# B&R Automation Studio project MotionTestBenchMaster (part 37)

#### Init.st - Init code
```iecst
PROGRAM _INIT
	(**********************************)
	(*  Mp Link Hierarchy management  *)
	(**********************************)
	fbMpComLinkToParent_Spare		(ParentLink := mpCOM_MAIN, MpLink := ADR(VAR_SpareLink));

	(**********************************)
	(* The machine is the higher Link *)
	(**********************************)
	fbMpComLinkToParent_Machine		(ParentLink := mpCOM_MAIN, MpLink := ADR(VAR_MachineLink));
	fbMpComLinkToParent_Master		(ParentLink := fbMpComLinkToParent_Machine.LinkOut,	MpLink := ADR(VAR_MasterModuleLink));
	fbMpComLinkToParent_Filler		(ParentLink := fbMpComLinkToParent_Machine.LinkOut,	MpLink := ADR(VAR_FillerModuleLink));

	IF VAR_AxOutletMain.nc_obj_inf.node_nr > 0 THEN	//At least the main axis in the outlet module
		fbMpComLinkToParent_Outlet	(ParentLink := fbMpComLinkToParent_Machine.LinkOut,	MpLink := ADR(VAR_OutletModuleLink));
	ELSE
		fbMpComLinkToParent_Outlet	(ParentLink := fbMpComLinkToParent_Spare.LinkOut,	MpLink := ADR(VAR_OutletModuleLink));
	END_IF

	IF VAR_AxInletMain.nc_obj_inf.node_nr > 0 THEN	//At least the main axis in the inlet module
		fbMpComLinkToParent_Inlet	(ParentLink := fbMpComLinkToParent_Machine.LinkOut,	MpLink := ADR(VAR_InletModuleLink));
	ELSE
		fbMpComLinkToParent_Inlet	(ParentLink := fbMpComLinkToParent_Spare.LinkOut,	MpLink := ADR(VAR_InletModuleLink));
	END_IF

	fbMpComLinkToParentAlarmMain	(ParentLink := fbMpComLinkToParent_Machine.LinkOut,	MpLink := ADR(gMainAlarmXCoreLink));

	(**********************************)
	(* Init of Link on Master Module  *)
	(**********************************)
	fbMpComLinkToParent_AlarmXMaster(ParentLink := fbMpComLinkToParent_Master.LinkOut,	MpLink := ADR(gMasterAlarmXCoreLink));
	fbMpComLinkToParent_MasterAxis 	(ParentLink := fbMpComLinkToParent_Master.LinkOut,	MpLink := ADR(gMasterLink));

	IF VAR_AxPowerSupply01.nc_obj_inf.node_nr > 0 THEN
		fbMpComLinkToParent_Pwr01 		(ParentLink := fbMpComLinkToParent_Master.LinkOut,	MpLink := ADR(gMasterPwr01Link));
	ELSE
		fbMpComLinkToParent_Pwr01		(ParentLink := fbMpComLinkToParent_Spare.LinkOut,	MpLink := ADR(gMasterPwr01Link));
	END_IF

	IF VAR_AxPowerSupply02.nc_obj_inf.node_nr > 0 THEN
		fbMpComLinkToParent_Pwr02 		(ParentLink := fbMpComLinkToParent_Master.LinkOut,	MpLink := ADR(gMasterPwr02Link));
	ELSE
		fbMpComLinkToParent_Pwr02 		(ParentLink := fbMpComLinkToParent_Spare.LinkOut,	MpLink := ADR(gMasterPwr02Link));
	END_IF

	(**********************************)
	(* Init of Link on Filler Module  *)
	(**********************************)
	fbMpComLinkToParent_AlarmXFiller(ParentLink := fbMpComLinkToParent_Filler.LinkOut,	MpLink := ADR(gFillerAlarmXCoreLink));
	fbMpComLinkToParent_FillerMas 	(ParentLink := fbMpComLinkToParent_Filler.LinkOut,	MpLink := ADR(gFillerModuleMasterLink));
	fbMpComLinkToParent_Carousel 	(ParentLink := fbMpComLinkToParent_Filler.LinkOut,	MpLink := ADR(gFillerMainLink));

	IF VAR_AxFillerIn01.nc_obj_inf.node_nr > 0 THEN
		fbMpComLinkToParent_FlrInlet01 	(ParentLink := fbMpComLinkToParent_Filler.LinkOut,	MpLink := ADR(gFlrIn01Link));
	ELSE
		fbMpComLinkToParent_FlrInlet01 	(ParentLink := fbMpComLinkToParent_Spare.LinkOut,	MpLink := ADR(gFlrIn01Link));
	END_IF

	IF VAR_AxFillerIn02.nc_obj_inf.node_nr > 0 THEN
		fbMpComLinkToParent_FlrInlet02 	(ParentLink := fbMpComLinkToParent_Filler.LinkOut,	MpLink := ADR(gFlrIn02Link));
	ELSE
		fbMpComLinkToParent_FlrInlet02 	(ParentLink := fbMpComLinkToParent_Spare.LinkOut,	MpLink := ADR(gFlrIn02Link));
	END_IF

	IF VAR_AxFillerIn03.nc_obj_inf.node_nr > 0 THEN
		fbMpComLinkToParent_FlrInlet03 	(ParentLink := fbMpComLinkToParent_Filler.LinkOut,	MpLink := ADR(gFlrIn03Link));
	ELSE
		fbMpComLinkToParent_FlrInlet03 	(ParentLink := fbMpComLinkToParent_Spare.LinkOut,	MpLink := ADR(gFlrIn03Link));
	END_IF

	IF VAR_AxFillerIn04.nc_obj_inf.node_nr > 0 THEN
		fbMpComLinkToParent_FlrInlet04 	(ParentLink := fbMpComLinkToParent_Filler.LinkOut,	MpLink := ADR(gFlrIn04Link));
	ELSE
		fbMpComLinkToParent_FlrInlet04 	(ParentLink := fbMpComLinkToParent_Spare.LinkOut,	MpLink := ADR(gFlrIn04Link));
	END_IF

	IF VAR_AxFillerIn05.nc_obj_inf.node_nr > 0 THEN
		fbMpComLinkToParent_FlrInlet05 	(ParentLink := fbMpComLinkToParent_Filler.LinkOut,	MpLink := ADR(gFlrIn05Link));
	ELSE
		fbMpComLinkToParent_FlrInlet05 	(ParentLink := fbMpComLinkToParent_Spare.LinkOut,	MpLink := ADR(gFlrIn05Link));
	END_IF

	IF VAR_AxFillerIn06.nc_obj_inf.node_nr > 0 THEN
		fbMpComLinkToParent_FlrInlet06 	(ParentLink := fbMpComLinkToParent_Filler.LinkOut,	MpLink := ADR(gFlrIn06Link));
	ELSE
		fbMpComLinkToParent_FlrInlet06 	(ParentLink := fbMpComLinkToParent_Spare.LinkOut,	MpLink := ADR(gFlrIn06Link));
	END_IF

	IF VAR_AxFillerIn07.nc_obj_inf.node_nr > 0 THEN
		fbMpComLinkToParent_FlrInlet07 	(ParentLink := fbMpComLinkToParent_Filler.LinkOut,	MpLink := ADR(gFlrIn07Link));
	ELSE
		fbMpComLinkToParent_FlrInlet07 	(ParentLink := fbMpComLinkToParent_Spare.LinkOut,	MpLink := ADR(gFlrIn07Link));
	END_IF

	IF VAR_AxFillerIn08.nc_obj_inf.node_nr > 0 THEN
		fbMpComLinkToParent_FlrInlet08 	(ParentLink := fbMpComLinkToParent_Filler.LinkOut,	MpLink := ADR(gFlrIn08Link));
	ELSE
		fbMpComLinkToParent_FlrInlet08 	(ParentLink := fbMpComLinkToParent_Spare.LinkOut,	MpLink := ADR(gFlrIn08Link));
	END_IF

	IF VAR_AxFillerIn09.nc_obj_inf.node_nr > 0 THEN
		fbMpComLinkToParent_FlrInlet09 	(ParentLink := fbMpComLinkToParent_Filler.LinkOut,	MpLink := ADR(gFlrIn09Link));
	ELSE
		fbMpComLinkToParent_FlrInlet09 	(ParentLink := fbMpComLinkToParent_Spare.LinkOut,	MpLink := ADR(gFlrIn09Link));
	END_IF

	IF VAR_AxFillerIn10.nc_obj_inf.node_nr > 0 THEN
		fbMpComLinkToParent_FlrInlet10 	(ParentLink := fbMpComLinkToParent_Filler.LinkOut,	MpLink := ADR(gFlrIn10Link));
	ELSE
		fbMpComLinkToParent_FlrInlet10 	(ParentLink := fbMpComLinkToParent_Spare.LinkOut,	MpLink := ADR(gFlrIn10Link));
	END_IF

	IF VAR_AxFillerOut01.nc_obj_inf.node_nr > 0 THEN
		fbMpComLinkToParent_FlrOutlet01	(ParentLink := fbMpComLinkToParent_Filler.LinkOut,	MpLink := ADR(gFlrOut01Link));
	ELSE
		fbMpComLinkToParent_FlrOutlet01 (ParentLink := fbMpComLinkToParent_Spare.LinkOut,	MpLink := ADR(gFlrOut01Link));
	END_IF

	IF VAR_AxFillerOut02.nc_obj_inf.node_nr > 0 THEN
		fbMpComLinkToParent_FlrOutlet02	(ParentLink := fbMpComLinkToParent_Filler.LinkOut,	MpLink := ADR(gFlrOut02Link));
	ELSE
		fbMpComLinkToParent_FlrOutlet02 (ParentLink := fbMpComLinkToParent_Spare.LinkOut,	MpLink := ADR(gFlrOut02Link));
	END_IF

	IF VAR_AxFillerOut03.nc_obj_inf.node_nr > 0 THEN
		fbMpComLinkToParent_FlrOutlet03	(ParentLink := fbMpComLinkToParent_Filler.LinkOut,	MpLink := ADR(gFlrOut03Link));
	ELSE
		fbMpComLinkToParent_FlrOutlet03 (ParentLink := fbMpComLinkToParent_Spare.LinkOut,	MpLink := ADR(gFlrOut03Link));
	END_IF

	IF VAR_AxFillerOut04.nc_obj_inf.node_nr > 0 THEN
		fbMpComLinkToParent_FlrOutlet04	(ParentLink := fbMpComLinkToParent_Filler.LinkOut,	MpLink := ADR(gFlrOut04Link));
	ELSE
		fbMpComLinkToParent_FlrOutlet04 (ParentLink := fbMpComLinkToParent_Spare.LinkOut,	MpLink := ADR(gFlrOut04Link));
	END_IF

	IF VAR_AxFillerOut05.nc_obj_inf.node_nr > 0 THEN
		fbMpComLinkToParent_FlrOutlet05	(ParentLink := fbMpComLinkToParent_Filler.LinkOut,	MpLink := ADR(gFlrOut05Link));
	ELSE
		fbMpComLinkToParent_FlrOutlet05 (ParentLink := fbMpComLinkToParent_Spare.LinkOut,	MpLink := ADR(gFlrOut05Link));
	END_IF

	IF VAR_AxFillerOut06.nc_obj_inf.node_nr > 0 THEN
		fbMpComLinkToParent_FlrOutlet06	(ParentLink := fbMpComLinkToParent_Filler.LinkOut,	MpLink := ADR(gFlrOut06Link));
	ELSE
		fbMpComLinkToParent_FlrOutlet06 (ParentLink := fbMpComLinkToParent_Spare.LinkOut,	MpLink := ADR(gFlrOut06Link));
	END_IF

	(**********************************)
	(* Init of Link on Inlet  Module  *)
	(**********************************)
	IF VAR_AxInletMain.nc_obj_inf.node_nr <> 0  THEN
		fbMpComLinkToParent_AlarmXInlet	(ParentLink := fbMpComLinkToParent_Inlet.LinkOut,	MpLink := ADR(gInletAlarmXCoreLink));
		fbMpComLinkToParent_InletMas 	(ParentLink := fbMpComLinkToParent_Inlet.LinkOut,	MpLink := ADR(gInletModuleMasterLink));
		fbMpComLinkToParent_InletMain	(ParentLink := fbMpComLinkToParent_Inlet.LinkOut,	MpLink := ADR(gInletMainLink));
	ELSE
		fbMpComLinkToParent_AlarmXInlet	(ParentLink := fbMpComLinkToParent_Spare.LinkOut,	MpLink := ADR(gInletAlarmXCoreLink));
		fbMpComLinkToParent_InletMas 	(ParentLink := fbMpComLinkToParent_Spare.LinkOut,	MpLink := ADR(gInletModuleMasterLink));
		fbMpComLinkToParent_InletMain	(ParentLink := fbMpComLinkToParent_Spare.LinkOut,	MpLink := ADR(gInletMainLink));
	END_IF

	(*  INLET 01 *)
	IF VAR_AxInletIn01.nc_obj_inf.node_nr <> 0 THEN
		fbMpComLinkToParent_InInlet01	(ParentLink := fbMpComLinkToParent_Inlet.LinkOut,	MpLink := ADR(gInInlet01Link));
	ELSE
		fbMpComLinkToParent_InInlet01 	(ParentLink := fbMpComLinkToParent_Spare.LinkOut,	MpLink := ADR(gInInlet01Link));
	END_IF

	(*  INLET 02 *)
	IF VAR_AxInletIn02.nc_obj_inf.node_nr <> 0 THEN
		fbMpComLinkToParent_InInlet02	(ParentLink := fbMpComLinkToParent_Inlet.LinkOut,	MpLink := ADR(gInInlet02Link));
	ELSE
		fbMpComLinkToParent_InInlet02 	(ParentLink := fbMpComLinkToParent_Spare.LinkOut,	MpLink := ADR(gInInlet02Link));
	END_IF

	(* INLET 03 *)
	IF VAR_AxInletIn03.nc_obj_inf.node_nr <> 0 THEN
		fbMpComLinkToParent_InInlet03	(ParentLink := fbMpComLinkToParent_Inlet.LinkOut,	MpLink := ADR(gInInlet03Link));
	ELSE
		fbMpComLinkToParent_InInlet03 	(ParentLink := fbMpComLinkToParent_Spare.LinkOut,	MpLink := ADR(gInInlet03Link));
	END_IF

	(* INLET 04*)
	IF VAR_AxInletIn04.nc_obj_inf.node_nr <> 0 THEN
		fbMpComLinkToParent_InInlet04	(ParentLink := fbMpComLinkToParent_Inlet.LinkOut,	MpLink := ADR(gInInlet04Link));
	ELSE
		fbMpComLinkToParent_InInlet04 	(ParentLink := fbMpComLinkToParent_Spare.LinkOut,	MpLink := ADR(gInInlet04Link));
	END_IF

	(*  OUTLET 01 *)
	IF VAR_AxInletOut01.nc_obj_inf.node_nr <> 0 THEN
		fbMpComLinkToParent_InOutlet01	(ParentLink := fbMpComLinkToParent_Inlet.LinkOut,	MpLink := ADR(gInOutlet01Link));
	ELSE
		fbMpComLinkToParent_InOutlet01 	(ParentLink := fbMpComLinkToParent_Spare.LinkOut,	MpLink := ADR(gInOutlet01Link));
	END_IF

	(*  OUTLET 02 *)
	IF VAR_AxInletOut02.nc_obj_inf.node_nr <> 0 THEN
		fbMpComLinkToParent_InOutlet02	(ParentLink := fbMpComLinkToParent_Inlet.LinkOut,	MpLink := ADR(gInOutlet02Link));
	ELSE
		fbMpComLinkToParent_InOutlet02 	(ParentLink := fbMpComLinkToParent_Spare.LinkOut,	MpLink := ADR(gInOutlet02Link));
	END_IF

	(* OUTLET 03 *)
	IF VAR_AxInletOut03.nc_obj_inf.node_nr <> 0 THEN
		fbMpComLinkToParent_InOutlet03	(ParentLink := fbMpComLinkToParent_Inlet.LinkOut,	MpLink := ADR(gInOutlet03Link));
	ELSE
		fbMpComLinkToParent_InOutlet03 	(ParentLink := fbMpComLinkToParent_Spare.LinkOut,	MpLink := ADR(gInOutlet03Link));
	END_IF

	(* OUTLET 04*)
	IF VAR_AxOutletOut04.nc_obj_inf.node_nr <> 0 THEN
		fbMpComLinkToParent_InOutlet04	(ParentLink := fbMpComLinkToParent_Inlet.LinkOut,	MpLink := ADR(gInOutlet04Link));
	ELSE
		fbMpComLinkToParent_InOutlet04 	(ParentLink := fbMpComLinkToParent_Spare.LinkOut,	MpLink := ADR(gInOutlet04Link));
	END_IF

	(**********************************)
	(* Init of Link on Outlet Module  *)
	(**********************************)
	IF VAR_AxOutletMain.nc_obj_inf.node_nr <> 0  THEN
		fbMpComLinkToParent_AlarmXOutlet(ParentLink := fbMpComLinkToParent_Outlet.LinkOut,	MpLink := ADR(gOutletAlarmXCoreLink));
		fbMpComLinkToParent_OutletMas 	(ParentLink := fbMpComLinkToParent_Outlet.LinkOut,	MpLink := ADR(gOutletModuleMasterLink));
		fbMpComLinkToParent_OutletMain	(ParentLink := fbMpComLinkToParent_Outlet.LinkOut,	MpLink := ADR(gOutletMainLink));
	ELSE
		fbMpComLinkToParent_AlarmXOutlet(ParentLink := fbMpComLinkToParent_Spare.LinkOut,	MpLink := ADR(gOutletAlarmXCoreLink));
		fbMpComLinkToParent_OutletMas 	(ParentLink := fbMpComLinkToParent_Spare.LinkOut,	MpLink := ADR(gOutletModuleMasterLink));
		fbMpComLinkToParent_OutletMain	(ParentLink := fbMpComLinkToParent_Spare.LinkOut,	MpLink := ADR(gOutletMainLink));
	END_IF

	(*  INLET 01 *)
	IF VAR_AxOutletIn01.nc_obj_inf.node_nr <> 0 THEN
		fbMpComLinkToParent_OutInlet01	(ParentLink := fbMpComLinkToParent_Outlet.LinkOut,	MpLink := ADR(gOutInlet01Link));
	ELSE
		fbMpComLinkToParent_OutInlet01 	(ParentLink := fbMpComLinkToParent_Spare.LinkOut,	MpLink := ADR(gOutInlet01Link));
	END_IF

	(*  INLET 02 *)
	IF VAR_AxOutletIn02.nc_obj_inf.node_nr <> 0 THEN
		fbMpComLinkToParent_OutInlet02	(ParentLink := fbMpComLinkToParent_Outlet.LinkOut,	MpLink := ADR(gOutInlet02Link));
	ELSE
		fbMpComLinkToParent_OutInlet02 	(ParentLink := fbMpComLinkToParent_Spare.LinkOut,	MpLink := ADR(gOutInlet02Link));
	END_IF

	(* INLET 03 *)
	IF VAR_AxOutletIn03.nc_obj_inf.node_nr <> 0 THEN
		fbMpComLinkToParent_OutInlet03	(ParentLink := fbMpComLinkToParent_Outlet.LinkOut,	MpLink := ADR(gOutInlet03Link));
	ELSE
		fbMpComLinkToParent_OutInlet03 	(ParentLink := fbMpComLinkToParent_Spare.LinkOut,	MpLink := ADR(gOutInlet03Link));
	END_IF

	(* INLET 04*)
	IF VAR_AxOutletIn04.nc_obj_inf.node_nr <> 0 THEN
		fbMpComLinkToParent_OutInlet04	(ParentLink := fbMpComLinkToParent_Outlet.LinkOut,	MpLink := ADR(gOutInlet04Link));
	ELSE
		fbMpComLinkToParent_OutInlet04 	(ParentLink := fbMpComLinkToParent_Spare.LinkOut,	MpLink := ADR(gOutInlet04Link));
	END_IF

	(*  OUTLET 01 *)
	IF VAR_AxOutletOut01.nc_obj_inf.node_nr <> 0 THEN
		fbMpComLinkToParent_OutOutlet01	(ParentLink := fbMpComLinkToParent_Outlet.LinkOut,	MpLink := ADR(gOutOutlet01Link));
	ELSE
		fbMpComLinkToParent_OutOutlet01 (ParentLink := fbMpComLinkToParent_Spare.LinkOut,	MpLink := ADR(gOutOutlet01Link));
	END_IF

	(*  OUTLET 02 *)
	IF VAR_AxOutletOut02.nc_obj_inf.node_nr <> 0 THEN
		fbMpComLinkToParent_OutOutlet02	(ParentLink := fbMpComLinkToParent_Outlet.LinkOut,	MpLink := ADR(gOutOutlet02Link));
	ELSE
		fbMpComLinkToParent_OutOutlet02 (ParentLink := fbMpComLinkToParent_Spare.LinkOut,	MpLink := ADR(gOutOutlet02Link));
	END_IF

	(* OUTLET 03 *)
	IF VAR_AxOutletOut03.nc_obj_inf.node_nr <> 0 THEN
		fbMpComLinkToParent_OutOutlet03	(ParentLink := fbMpComLinkToParent_Outlet.LinkOut,	MpLink := ADR(gOutOutlet03Link));
	ELSE
		fbMpComLinkToParent_OutOutlet03 (ParentLink := fbMpComLinkToParent_Spare.LinkOut,	MpLink := ADR(gOutOutlet03Link));
	END_IF

	(* OUTLET 04*)
	IF VAR_AxOutletOut04.nc_obj_inf.node_nr <> 0 THEN
		fbMpComLinkToParent_OutOutlet04	(ParentLink := fbMpComLinkToParent_Outlet.LinkOut,	MpLink := ADR(gOutOutlet04Link));
	ELSE
		fbMpComLinkToParent_OutOutlet04 (ParentLink := fbMpComLinkToParent_Spare.LinkOut,	MpLink := ADR(gOutOutlet04Link));
	END_IF
END_PROGRAM

PROGRAM _CYCLIC
	ST_tmp_suspend(0);
END_PROGRAM
```

#### Variables.var - Local variables
```iecst
(*Link To Parent Machine*)
VAR
	fbMpComLinkToParent_Machine : MpComLinkToParent;
	fbMpComLinkToParent_Spare : MpComLinkToParent;
	fbMpComLinkToParentAlarmMain : MpComLinkToParent;
END_VAR
(*Link To Paret Master Module*)
VAR
	fbMpComLinkToParent_Master : MpComLinkToParent;
	fbMpComLinkToParent_Pwr01 : MpComLinkToParent;
	fbMpComLinkToParent_Pwr02 : MpComLinkToParent;
	fbMpComLinkToParent_MasterAxis : MpComLinkToParent;
	fbMpComLinkToParent_AlarmXMaster : MpComLinkToParent;
END_VAR
(*Link To Paret Filler Module*)
VAR
	fbMpComLinkToParent_Filler : MpComLinkToParent;
	fbMpComLinkToParent_FillerMas : MpComLinkToParent;
	fbMpComLinkToParent_Carousel : MpComLinkToParent;
	fbMpComLinkToParent_FlrInlet01 : MpComLinkToParent;
	fbMpComLinkToParent_FlrInlet02 : MpComLinkToParent;
	fbMpComLinkToParent_FlrInlet03 : MpComLinkToParent;
	fbMpComLinkToParent_FlrInlet04 : MpComLinkToParent;
	fbMpComLinkToParent_FlrInlet05 : MpComLinkToParent;
	fbMpComLinkToParent_FlrInlet06 : MpComLinkToParent;
	fbMpComLinkToParent_FlrInlet07 : MpComLinkToParent;
	fbMpComLinkToParent_FlrInlet08 : MpComLinkToParent;
	fbMpComLinkToParent_FlrInlet09 : MpComLinkToParent;
	fbMpComLinkToParent_FlrInlet10 : MpComLinkToParent;
	fbMpComLinkToParent_FlrOutlet01 : MpComLinkToParent;
	fbMpComLinkToParent_FlrOutlet02 : MpComLinkToParent;
	fbMpComLinkToParent_FlrOutlet03 : MpComLinkToParent;
	fbMpComLinkToParent_FlrOutlet04 : MpComLinkToParent;
	fbMpComLinkToParent_FlrOutlet05 : MpComLinkToParent;
	fbMpComLinkToParent_FlrOutlet06 : MpComLinkToParent;
	fbMpComLinkToParent_AlarmXFiller : MpComLinkToParent;
END_VAR
(*Link To Paret Inlet Module*)
VAR
	fbMpComLinkToParent_Inlet : MpComLinkToParent;
	fbMpComLinkToParent_InletMas : MpComLinkToParent;
	fbMpComLinkToParent_InletMain : MpComLinkToParent;
	fbMpComLinkToParent_InInlet01 : MpComLinkToParent;
	fbMpComLinkToParent_InInlet02 : MpComLinkToParent;
	fbMpComLinkToParent_InInlet03 : MpComLinkToParent;
	fbMpComLinkToParent_InInlet04 : MpComLinkToParent;
	fbMpComLinkToParent_InOutlet01 : MpComLinkToParent;
	fbMpComLinkToParent_InOutlet02 : MpComLinkToParent;
	fbMpComLinkToParent_InOutlet03 : MpComLinkToParent;
	fbMpComLinkToParent_InOutlet04 : MpComLinkToParent;
	fbMpComLinkToParent_AlarmXInlet : MpComLinkToParent;
END_VAR
(*Link To Paret Outlet Module*)
VAR
	fbMpComLinkToParent_Outlet : MpComLinkToParent;
	fbMpComLinkToParent_OutletMas : MpComLinkToParent;
	fbMpComLinkToParent_OutletMain : MpComLinkToParent;
	fbMpComLinkToParent_OutInlet01 : MpComLinkToParent;
	fbMpComLinkToParent_OutInlet02 : MpComLinkToParent;
	fbMpComLinkToParent_OutInlet03 : MpComLinkToParent;
	fbMpComLinkToParent_OutInlet04 : MpComLinkToParent;
	fbMpComLinkToParent_OutOutlet01 : MpComLinkToParent;
	fbMpComLinkToParent_OutOutlet02 : MpComLinkToParent;
	fbMpComLinkToParent_OutOutlet03 : MpComLinkToParent;
	fbMpComLinkToParent_OutOutlet04 : MpComLinkToParent;
	fbMpComLinkToParent_AlarmXOutlet : MpComLinkToParent;
END_VAR
```

### Program Logical/30_MC/Task/Cyclic01/MC_FAST (IEC) - MC_FAST - C#1 (0.8ms)

#### Variables.var
```iecst
(*Master MC Version*)
VAR
	diMachineModuloPos : DINT;
	diInletModuloPos : DINT;
	diFillerModuloPos : DINT;
	diOutletModuloPos : DINT;
END_VAR
(*Virtual position cyclic read*)
VAR
	fbReadCyclicParID : ARRAY[0..3] OF MC_BR_InitCyclicRead;
END_VAR
(*Cam*)
VAR
	fbCamMachineCkAB : FB_CamGeneratorAB_v2;
	fbCam01 : FB_CamGenerator_v2;
	fbCam02 : FB_CamGenerator_v2;
	fbCam03 : FB_CamGenerator_v2;
	fbCam04 : FB_CamGenerator_v2;
	fbCam05 : FB_CamGenerator_v2;
	fbCam06 : FB_CamGenerator_v2;
	fbCam07 : FB_CamGenerator_v2;
	fbCam08 : FB_CamGenerator_v2;
	fbCam09 : FB_CamGenerator_v2;
	fbCam10 : FB_CamGenerator_v2;
	fbCam11 : FB_CamGenerator_v2; (*v999 test*)
END_VAR
(*Auxiliary*)
VAR
	xDummy : BOOL;
	xAutoModActive : BOOL; (*V4.A.A.1.6.12i*)
	xMultiModActive : BOOL; (*V4.A.A.1.6.12i*)
END_VAR
```

#### Cyclic.sfc
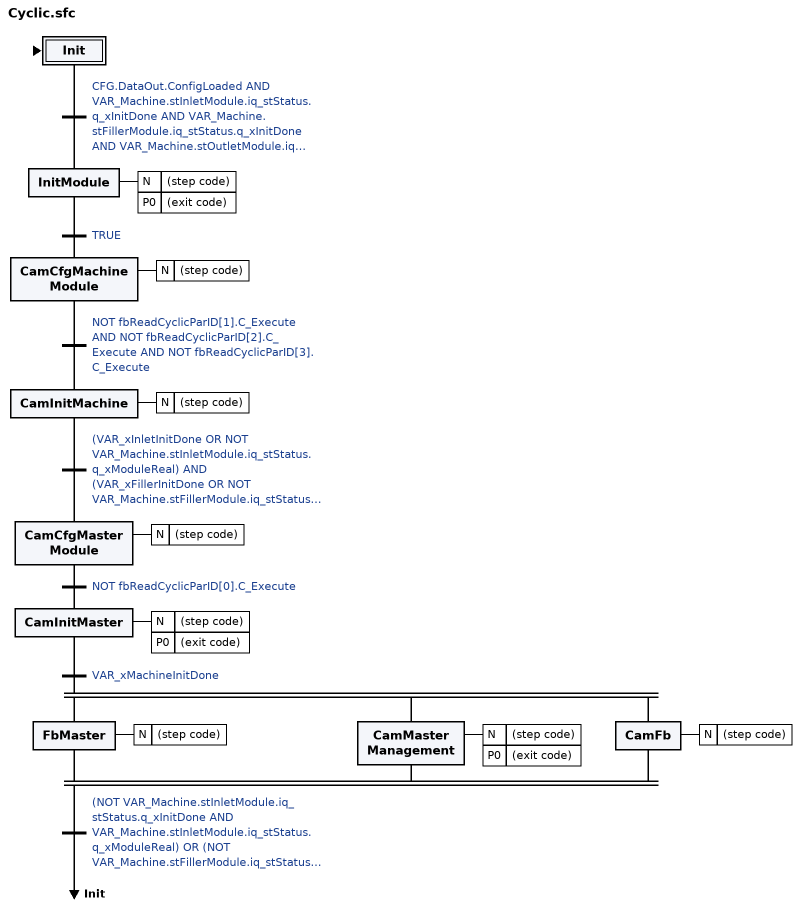
```iecst
PROGRAM _CYCLIC
INITIAL_STEP Init:
END_STEP
TRANSITION Configuration Loaded FROM Init TO InitModule:=
CFG.DataOut.ConfigLoaded AND
VAR_Machine.stInletModule.iq_stStatus.q_xInitDone	AND
VAR_Machine.stFillerModule.iq_stStatus.q_xInitDone	AND
VAR_Machine.stOutletModule.iq_stStatus.q_xInitDone
END_TRANSITION
STEP InitModule:
(*MACHINE MASTER AXIS*)
fbMachineMasterFast.i_xEnable					:= TRUE;	//V4.A.A.1.6.10
fbMachineMasterFast.i_pAxisADR 					:= ADR(VAR_AxMachineMaster);	//V4.A.A.1.6.10
fbMachineMasterFast.i_pstCmd					:= ADR(VAR_Machine.stMasterModule.iq_astSubModuleAxis[CST_MachineMasterAxis].iq_stCmd);	//V4.A.A.1.6.10
fbMachineMasterFast.i_pstParameter				:= ADR(VAR_Machine.stMasterModule.iq_astSubModuleAxis[CST_MachineMasterAxis].iq_stParam);	//V4.A.A.1.6.10
fbMachineMasterFast.i_pstStatus					:= ADR(VAR_Machine.stMasterModule.iq_astSubModuleAxis[CST_MachineMasterAxis].iq_stStatus);	//V4.A.A.1.6.10
fbMachineMasterFast.i_pstAxisHome				:= ADR(VAR_AxMachineMasterHomeData);	//V4.A.A.1.6.10

// Only for machine master
fbMachineMasterFast.i_pstAbsEncPerm				:= ADR(VAR_AbsEncPerm);	//V4.A.A.1.6.10
fbMachineMasterFast.i_xCmdEnableCurves			:= FALSE;	//V4.A.A.1.6.10

IF CFG_MC.Generic.SyncroPar.ExternalEncoder THEN	//V4.A.A.1.6.10(COMBI with encoder*)
	fbMachineMasterFast.i_xExternalEncoder			:= TRUE;	//V4.A.A.1.6.10
	fbMachineMasterFast.i_uiFilteringCoefficient	:= CST_ExtEncFilteringCoefficient;	//V4.A.A.1.6.10
	fbMachineMasterFast.i_uiNumberOfEplCycles		:= CST_ExtEncNumberOfExtCycles;	//V4.A.A.1.6.10
ELSE	//V4.A.A.1.6.10          (*SSC*)
	fbMachineMasterFast.i_xExternalEncoder			:= FALSE;	//V4.A.A.1.6.10
	fbMachineMasterFast.i_xExternalPositionFormat	:= CFG_MC.Generic.SyncroPar.ExternalPositionFormat;//v4.A.A.1.7.0
	fbMachineMasterFast.i_uiFilteringCoefficient	:= CST_FilteringCoefficient;	//V4.A.A.1.6.10
	fbMachineMasterFast.i_uiNumberOfEplCycles		:= CST_NumberOfExtCycles;	//V4.A.A.1.6.10
END_IF	//V4.A.A.1.6.10

fbMachineMasterFast.i_uiNumberOfSteps			:= CFG_MC.Generic.SyncroPar.NumberOfSteps;	//V4.A.A.1.6.10
fbMachineMasterFast.i_udiExternalSignalPeriod	:= CFG_MC.Generic.SyncroPar.ExternalSignalPeriod;	//V4.A.A.1.6.10
END_STEP
EXIT_ACTION
IF CFG_MC.Generic.SyncroPar.ExternalPositionFormat THEN//v4.A.A.1.7.0
	fbMachineMasterFast.i_pstExtEncoderPosition		:= ITC.DataOut.AdrExternalPosition;//v4.A.A.1.7.0
ELSE//v4.A.A.1.7.0
	fbMachineMasterFast.i_pstExtEncoderPosition		:= ADR(ITC_Motion_ExtEnc);//v4.A.A.1.7.0
END_IF//v4.A.A.1.7.0

//fbMachineMasterFast.i_pstExtEncoderPosition		:= ADR(ITC_Motion_ExtEnc);	//V4.A.A.1.6.10
fbMachineMasterFast.i_pstMasterPositionStruct	:= VAR_Machine.stMasterModule.iq_stParameters.i_pstMasterPositionStruct;	//V4.A.A.1.6.10
END_ACTION
TRANSITION FROM InitModule TO CamCfgMachineModule:=
TRUE
END_TRANSITION
STEP CamCfgMachineModule:
(* Initialization of cyclic position reading for Inlet module *)
fbReadCyclicParID[1].Axis			:= ADR(VAR_AxInletModuleMaster);
fbReadCyclicParID[1].DataAddress	:= ADR(diInletModuloPos);
fbReadCyclicParID[1].DataType		:= ncPAR_TYP_DINT;
fbReadCyclicParID[1].ParID			:= ACP10PAR_CURVE_VALUE_REL_I4 + 5;

(* Initialization of cyclic position reading for Filler module *)
fbReadCyclicParID[2].Axis			:= ADR(VAR_AxFillerModuleMaster);
fbReadCyclicParID[2].DataAddress	:= ADR(diFillerModuloPos);
fbReadCyclicParID[2].DataType		:= ncPAR_TYP_DINT;
fbReadCyclicParID[2].ParID			:= ACP10PAR_CURVE_VALUE_REL_I4 + 5;

(* Initialization of cyclic position reading for Outlet module *)
fbReadCyclicParID[3].Axis			:= ADR(VAR_AxOutletModuleMaster);
fbReadCyclicParID[3].DataAddress	:= ADR(diOutletModuloPos);
fbReadCyclicParID[3].DataType		:= ncPAR_TYP_DINT;
fbReadCyclicParID[3].ParID			:= ACP10PAR_CURVE_VALUE_REL_I4 + 5;

//V4.A.A.1.6.12d
VAR_xMachineInitDone	:= FALSE;
VAR_xInletInitDone		:= FALSE;
VAR_xFillerInitDone		:= FALSE;
VAR_xOutletInitDone		:= FALSE;

fbReadCyclicParID[1].Execute := FALSE;//V4.A.A.1.6.12d
fbReadCyclicParID[2].Execute := FALSE;//V4.A.A.1.6.12d
fbReadCyclicParID[3].Execute := FALSE;//V4.A.A.1.6.12d

fbReadCyclicParID[1]();//V4.A.A.1.6.12d
fbReadCyclicParID[2]();//V4.A.A.1.6.12d
fbReadCyclicParID[3]();//V4.A.A.1.6.12d
END_STEP
TRANSITION CamConfiguredMachine FROM CamCfgMachineModule TO CamInitMachine:=
NOT fbReadCyclicParID[1].C_Execute AND
NOT fbReadCyclicParID[2].C_Execute AND
NOT fbReadCyclicParID[3].C_Execute //V4.A.A.1.6.12d
END_TRANSITION
STEP CamInitMachine:
(* Initialization of cyclic position reading for Inlet module *)
IF VAR_Machine.stInletModule.iq_stStatus.q_xModuleReal THEN
	IF NOT VAR_xInletInitDone THEN
		IF NOT fbReadCyclicParID[1].Execute THEN
			fbReadCyclicParID[1].Execute	:= TRUE;
		ELSE
			IF fbReadCyclicParID[1].Done OR fbReadCyclicParID[1].Error THEN
				VAR_xInletInitDone := TRUE;
				fbReadCyclicParID[1].Execute := FALSE;//1.7.2a
			END_IF
		END_IF
	ELSE
		fbReadCyclicParID[1].Execute := FALSE;
	END_IF
ELSE
	VAR_xInletInitDone := TRUE;
END_IF

IF fbReadCyclicParID[1].Execute OR fbReadCyclicParID[1].Busy THEN
	fbReadCyclicParID[1]();
END_IF

(* Initialization of cyclic position reading for Filler module *)
IF VAR_Machine.stFillerModule.iq_stStatus.q_xModuleReal THEN
	IF NOT VAR_xFillerInitDone THEN
		IF NOT fbReadCyclicParID[2].Execute THEN
			fbReadCyclicParID[2].Execute	:= TRUE;
		ELSE
			IF fbReadCyclicParID[2].Done OR fbReadCyclicParID[2].Error THEN
				VAR_xFillerInitDone := TRUE;
				fbReadCyclicParID[2].Execute := FALSE;//1.7.2a
			END_IF
		END_IF
	ELSE
		fbReadCyclicParID[2].Execute := FALSE;
	END_IF
ELSE
	VAR_xFillerInitDone := TRUE;
END_IF

IF fbReadCyclicParID[2].Execute OR fbReadCyclicParID[2].Busy THEN
	fbReadCyclicParID[2]();
END_IF

(* Initialization of cyclic position reading for Outlet module *)
IF VAR_Machine.stOutletModule.iq_stStatus.q_xModuleReal THEN
	IF NOT VAR_xOutletInitDone THEN
		IF NOT fbReadCyclicParID[3].Execute THEN
			fbReadCyclicParID[3].Execute	:= TRUE;
		ELSE
			IF fbReadCyclicParID[3].Done OR fbReadCyclicParID[3].Error THEN
				VAR_xOutletInitDone := TRUE;
				fbReadCyclicParID[3].Execute := FALSE;//1.7.2a
			END_IF
		END_IF
	ELSE
		fbReadCyclicParID[3].Execute := FALSE;
	END_IF
ELSE
	VAR_xOutletInitDone := TRUE;
END_IF

IF fbReadCyclicParID[3].Execute OR fbReadCyclicParID[3].Busy THEN
	fbReadCyclicParID[3]();
END_IF
END_STEP
TRANSITION Cam Initialized Machine FROM CamInitMachine TO CamCfgMasterModule:=
(VAR_xInletInitDone		OR NOT VAR_Machine.stInletModule.iq_stStatus.q_xModuleReal) AND
(VAR_xFillerInitDone	OR NOT VAR_Machine.stFillerModule.iq_stStatus.q_xModuleReal) AND
(VAR_xOutletInitDone	OR NOT VAR_Machine.stOutletModule.iq_stStatus.q_xModuleReal) AND
VAR_Machine.stMasterModule.iq_astSubModuleAxis[0].iq_stStatus.q_stMainAxisStatus.q_xInitDone
END_TRANSITION
STEP CamCfgMasterModule:
//V4.A.A.1.6.12d new position
(* Initialization of cyclic position reading for Master module *)
fbReadCyclicParID[0].Axis			:= ADR(VAR_AxMachineMaster);
fbReadCyclicParID[0].DataAddress	:= ADR(diMachineModuloPos);
fbReadCyclicParID[0].DataType		:= ncPAR_TYP_DINT;
fbReadCyclicParID[0].Mode			:= mcEVERY_RECORD; // V 1.1
fbReadCyclicParID[0].ParID			:= ACP10PAR_CURVE_VALUE_REL_I4 + 5;

fbReadCyclicParID[0].Execute := FALSE;//V4.A.A.1.6.12d

fbReadCyclicParID[0]();//V4.A.A.1.6.12d
END_STEP
TRANSITION CamConfiguredMaster FROM CamCfgMasterModule TO CamInitMaster:=
NOT fbReadCyclicParID[0].C_Execute
END_TRANSITION
STEP CamInitMaster:
(* Initialization of cyclic position reading for Master module *)
IF NOT VAR_xMachineInitDone THEN
	IF NOT fbReadCyclicParID[0].Execute THEN
		fbReadCyclicParID[0].Execute	:= TRUE;
	ELSE
		IF fbReadCyclicParID[0].Done OR fbReadCyclicParID[0].Error THEN
			VAR_xMachineInitDone := TRUE;
			fbReadCyclicParID[0].Execute := FALSE;//1.7.2a
		END_IF
	END_IF
ELSE
	fbReadCyclicParID[0].Execute := FALSE;
END_IF

IF fbReadCyclicParID[0].Execute OR fbReadCyclicParID[0].Busy THEN
	fbReadCyclicParID[0]();
END_IF
END_STEP
EXIT_ACTION
IF CFG_MC.Generic.Aseptic THEN
	fbCamMachineCkAB.i_rOnPositionA		:= CST_OnPositionCkA_Fma;
	fbCamMachineCkAB.i_rOffPositionA	:= CST_OffPositionCkA_Fma;
	fbCamMachineCkAB.i_rOnPositionB		:= CST_OnPositionCkB_Fma;
	fbCamMachineCkAB.i_rOffPositionB	:= CST_OffPositionCkB_Fma;
ELSE
	fbCamMachineCkAB.i_rOnPositionA		:= CST_OnPositionCkA;
	fbCamMachineCkAB.i_rOffPositionA	:= CST_OffPositionCkA;
	fbCamMachineCkAB.i_rOnPositionB		:= CST_OnPositionCkB;
	fbCamMachineCkAB.i_rOffPositionB	:= CST_OffPositionCkB;
END_IF
fbCamMachineCkAB.i_rAdvanceTime			:= CST_AdvTimeCkA;
fbCamMachineCkAB.i_pxPointerStepAdvA	:= ADR(xDummy);
fbCamMachineCkAB.i_pxPointerStepAdvB	:= ADR(xDummy);

fbCamMachineCkAB.i_pdiAxisPosition	:= ADR(diMachineModuloPos);
fbCamMachineCkAB.i_prAxisVelocity	:= ADR(VAR_AxMachineMaster.monitor.v);

fbCam01.i_pdiAxisPosition			:= ADR(diMachineModuloPos);
fbCam01.i_prAxisVelocity			:= ADR(VAR_AxMachineMaster.monitor.v);

fbCam02.i_pdiAxisPosition			:= ADR(diMachineModuloPos);
fbCam02.i_prAxisVelocity			:= ADR(VAR_AxMachineMaster.monitor.v);

fbCam03.i_pdiAxisPosition			:= ADR(diMachineModuloPos);
fbCam03.i_prAxisVelocity			:= ADR(VAR_AxMachineMaster.monitor.v);

fbCam04.i_pdiAxisPosition			:= ADR(diMachineModuloPos);
fbCam04.i_prAxisVelocity			:= ADR(VAR_AxMachineMaster.monitor.v);

fbCam05.i_pdiAxisPosition			:= ADR(diMachineModuloPos);
fbCam05.i_prAxisVelocity			:= ADR(VAR_AxMachineMaster.monitor.v);

fbCam06.i_pdiAxisPosition			:= ADR(diMachineModuloPos);
fbCam06.i_prAxisVelocity			:= ADR(VAR_AxMachineMaster.monitor.v);

fbCam07.i_pdiAxisPosition			:= ADR(diMachineModuloPos);
fbCam07.i_prAxisVelocity			:= ADR(VAR_AxMachineMaster.monitor.v);

fbCam08.i_pdiAxisPosition			:= ADR(diMachineModuloPos);
fbCam08.i_prAxisVelocity			:= ADR(VAR_AxMachineMaster.monitor.v);

fbCam09.i_pdiAxisPosition			:= ADR(diMachineModuloPos);
fbCam09.i_prAxisVelocity			:= ADR(VAR_AxMachineMaster.monitor.v);

fbCam10.i_pdiAxisPosition			:= ADR(diMachineModuloPos);
fbCam10.i_prAxisVelocity			:= ADR(VAR_AxMachineMaster.monitor.v);

fbCam11.i_pdiAxisPosition			:= ADR(diMachineModuloPos); //v999 test
fbCam11.i_prAxisVelocity			:= ADR(VAR_AxMachineMaster.monitor.v); //v999 test

VAR_CamInitialized	:= TRUE;
END_ACTION
TRANSITION Cam Initialized Master FROM CamInitMaster TO (FbMaster,CamMasterManagement,CamFb):=
VAR_xMachineInitDone
END_TRANSITION
STEP FbMaster:
fbMachineMasterFast;	//V4.A.A.1.6.10
END_STEP
STEP CamMasterManagement:
IF MC_InputOutput.Network.Machine.Status.MultiModalityActive AND NOT xMultiModActive THEN//V4.A.A.1.6.12i
	fbCamMachineCkAB.i_pdiAxisPosition	:= ADR(diFillerModuloPos);
	fbCamMachineCkAB.i_prAxisVelocity	:= ADR(VAR_AxFillerMain.monitor.v);

	fbCam01.i_pdiAxisPosition			:= ADR(diFillerModuloPos);
	fbCam01.i_prAxisVelocity			:= ADR(VAR_AxFillerMain.monitor.v);

	fbCam02.i_pdiAxisPosition			:= ADR(diFillerModuloPos);
	fbCam02.i_prAxisVelocity			:= ADR(VAR_AxFillerMain.monitor.v);

	fbCam03.i_pdiAxisPosition			:= ADR(diFillerModuloPos);
	fbCam03.i_prAxisVelocity			:= ADR(VAR_AxFillerMain.monitor.v);

	fbCam04.i_pdiAxisPosition			:= ADR(diFillerModuloPos);
	fbCam04.i_prAxisVelocity			:= ADR(VAR_AxFillerMain.monitor.v);

	fbCam05.i_pdiAxisPosition			:= ADR(diFillerModuloPos);
	fbCam05.i_prAxisVelocity			:= ADR(VAR_AxFillerMain.monitor.v);

	fbCam06.i_pdiAxisPosition			:= ADR(diFillerModuloPos);
	fbCam06.i_prAxisVelocity			:= ADR(VAR_AxFillerMain.monitor.v);

	fbCam07.i_pdiAxisPosition			:= ADR(diFillerModuloPos);
	fbCam07.i_prAxisVelocity			:= ADR(VAR_AxFillerMain.monitor.v);

	fbCam08.i_pdiAxisPosition			:= ADR(diFillerModuloPos);
	fbCam08.i_prAxisVelocity			:= ADR(VAR_AxFillerMain.monitor.v);

	IF VAR_Machine.stOutletModule.iq_stStatus.q_xModuleReal THEN
		fbCam09.i_pdiAxisPosition			:= ADR(VAR_AxOutletMain.monitor.s);
		fbCam09.i_prAxisVelocity			:= ADR(VAR_AxOutletMain.monitor.v);

		fbCam10.i_pdiAxisPosition			:= ADR(VAR_AxOutletMain.monitor.s);
		fbCam10.i_prAxisVelocity			:= ADR(VAR_AxOutletMain.monitor.v);
	ELSE
		fbCam09.i_pdiAxisPosition			:= ADR(diFillerModuloPos);
		fbCam09.i_prAxisVelocity			:= ADR(VAR_AxFillerMain.monitor.v);

		fbCam10.i_pdiAxisPosition			:= ADR(diFillerModuloPos);
		fbCam10.i_prAxisVelocity			:= ADR(VAR_AxFillerMain.monitor.v);
	END_IF

	fbCam11.i_pdiAxisPosition			:= ADR(diFillerModuloPos); //v999 test
	fbCam11.i_prAxisVelocity			:= ADR(VAR_AxFillerMain.monitor.v); //v999 test

	xMultiModActive := TRUE; //V4.A.A.1.6.12i
	xAutoModActive 	:= FALSE;//V4.A.A.1.6.12i

ELSIF NOT MC_InputOutput.Network.Machine.Status.MultiModalityActive AND NOT xAutoModActive THEN//V4.A.A.1.6.12i
	fbCamMachineCkAB.i_pdiAxisPosition	:= ADR(diMachineModuloPos);
	fbCamMachineCkAB.i_prAxisVelocity	:= ADR(VAR_AxMachineMaster.monitor.v);

	fbCam01.i_pdiAxisPosition			:= ADR(diMachineModuloPos);
	fbCam01.i_prAxisVelocity			:= ADR(VAR_AxMachineMaster.monitor.v);

	fbCam02.i_pdiAxisPosition			:= ADR(diMachineModuloPos);
	fbCam02.i_prAxisVelocity			:= ADR(VAR_AxMachineMaster.monitor.v);

	fbCam03.i_pdiAxisPosition			:= ADR(diMachineModuloPos);
	fbCam03.i_prAxisVelocity			:= ADR(VAR_AxMachineMaster.monitor.v);

	fbCam04.i_pdiAxisPosition			:= ADR(diMachineModuloPos);
	fbCam04.i_prAxisVelocity			:= ADR(VAR_AxMachineMaster.monitor.v);

	fbCam05.i_pdiAxisPosition			:= ADR(diMachineModuloPos);
	fbCam05.i_prAxisVelocity			:= ADR(VAR_AxMachineMaster.monitor.v);

	fbCam06.i_pdiAxisPosition			:= ADR(diMachineModuloPos);
	fbCam06.i_prAxisVelocity			:= ADR(VAR_AxMachineMaster.monitor.v);

	fbCam07.i_pdiAxisPosition			:= ADR(diMachineModuloPos);
	fbCam07.i_prAxisVelocity			:= ADR(VAR_AxMachineMaster.monitor.v);

	fbCam08.i_pdiAxisPosition			:= ADR(diMachineModuloPos);
	fbCam08.i_prAxisVelocity			:= ADR(VAR_AxMachineMaster.monitor.v);

	fbCam09.i_pdiAxisPosition			:= ADR(diMachineModuloPos);
	fbCam09.i_prAxisVelocity			:= ADR(VAR_AxMachineMaster.monitor.v);

	fbCam10.i_pdiAxisPosition			:= ADR(diMachineModuloPos);
	fbCam10.i_prAxisVelocity			:= ADR(VAR_AxMachineMaster.monitor.v);

	fbCam11.i_pdiAxisPosition			:= ADR(diMachineModuloPos); //v999 test
	fbCam11.i_prAxisVelocity			:= ADR(VAR_AxMachineMaster.monitor.v); //v999 test

	xMultiModActive := FALSE;//V4.A.A.1.6.12i
	xAutoModActive 	:= TRUE;//V4.A.A.1.6.12i
END_IF
END_STEP
EXIT_ACTION
VAR_CamInitialized := FALSE;
(* TODO: Insert Program *)
END_ACTION
STEP CamFb:
fbCamMachineCkAB(
i_xEnable			:= TRUE,
i_pxPointerOutputA	:= ADR(MC_InputOutput.Network.Machine.Status.MachineClockA),
i_pxPointerOutputB	:= ADR(MC_InputOutput.Network.Machine.Status.MachineClockB),
);

fbCam01(
i_xEnable			:= TRUE,
i_pxPointerOutput	:= ADR(MC_InputOutput.Network.Machine.Status.Clock01),
i_pxPointerStepAdv	:= ADR(MC_InputOutput.Network.Machine.Status.Clock01AdvStep),
i_rOnPosition		:= MC_InputOutput.Network.Machine.Parameters.Cam01OnValue,
i_rOffPosition		:= MC_InputOutput.Network.Machine.Parameters.Cam01OffValue,
i_rAdvanceTime		:= MC_InputOutput.Network.Machine.Parameters.Cam01AdvTime,
i_usiNumberOfPulse	:= MC_InputOutput.Network.Machine.Parameters.Cam01Pulse,
);

fbCam02(
i_xEnable			:= TRUE,
i_pxPointerOutput	:= ADR(MC_InputOutput.Network.Machine.Status.Clock02),
i_pxPointerStepAdv	:= ADR(MC_InputOutput.Network.Machine.Status.Clock02AdvStep),
i_rOnPosition		:= MC_InputOutput.Network.Machine.Parameters.Cam02OnValue,
i_rOffPosition		:= MC_InputOutput.Network.Machine.Parameters.Cam02OffValue,
i_rAdvanceTime		:= MC_InputOutput.Network.Machine.Parameters.Cam02AdvTime,
i_usiNumberOfPulse	:= MC_InputOutput.Network.Machine.Parameters.Cam02Pulse,
);

fbCam03(
i_xEnable			:= TRUE,
i_pxPointerOutput	:= ADR(MC_InputOutput.Network.Machine.Status.Clock03),
i_pxPointerStepAdv	:= ADR(MC_InputOutput.Network.Machine.Status.Clock03AdvStep),
i_rOnPosition		:= MC_InputOutput.Network.Machine.Parameters.Cam03OnValue,
i_rOffPosition		:= MC_InputOutput.Network.Machine.Parameters.Cam03OffValue,
i_rAdvanceTime		:= MC_InputOutput.Network.Machine.Parameters.Cam03AdvTime,
i_usiNumberOfPulse	:= MC_InputOutput.Network.Machine.Parameters.Cam03Pulse,
);

fbCam04(
i_xEnable			:= TRUE,
i_pxPointerOutput	:= ADR(MC_InputOutput.Network.Machine.Status.Clock04),
i_pxPointerStepAdv	:= ADR(MC_InputOutput.Network.Machine.Status.Clock04AdvStep),
i_rOnPosition		:= MC_InputOutput.Network.Machine.Parameters.Cam04OnValue,
i_rOffPosition		:= MC_InputOutput.Network.Machine.Parameters.Cam04OffValue,
i_rAdvanceTime		:= MC_InputOutput.Network.Machine.Parameters.Cam04AdvTime,
i_usiNumberOfPulse	:= MC_InputOutput.Network.Machine.Parameters.Cam04Pulse,
);

fbCam05(
i_xEnable			:= TRUE,
i_pxPointerOutput	:= ADR(MC_InputOutput.Network.Machine.Status.Clock05),
i_pxPointerStepAdv	:= ADR(MC_InputOutput.Network.Machine.Status.Clock05AdvStep),
i_rOnPosition		:= MC_InputOutput.Network.Machine.Parameters.Cam05OnValue,
i_rOffPosition		:= MC_InputOutput.Network.Machine.Parameters.Cam05OffValue,
i_rAdvanceTime		:= MC_InputOutput.Network.Machine.Parameters.Cam05AdvTime,
i_usiNumberOfPulse	:= MC_InputOutput.Network.Machine.Parameters.Cam05Pulse,
);

fbCam06(
i_xEnable			:= TRUE,
i_pxPointerOutput	:= ADR(MC_InputOutput.Network.Machine.Status.Clock06),
i_pxPointerStepAdv	:= ADR(MC_InputOutput.Network.Machine.Status.Clock06AdvStep),
i_rOnPosition		:= MC_InputOutput.Network.Machine.Parameters.Cam06OnValue,
i_rOffPosition		:= MC_InputOutput.Network.Machine.Parameters.Cam06OffValue,
i_rAdvanceTime		:= MC_InputOutput.Network.Machine.Parameters.Cam06AdvTime,
i_usiNumberOfPulse	:= MC_InputOutput.Network.Machine.Parameters.Cam06Pulse,
);

fbCam07(
i_xEnable			:= TRUE,
i_pxPointerOutput	:= ADR(MC_InputOutput.Network.Machine.Status.Clock07),
i_pxPointerStepAdv	:= ADR(MC_InputOutput.Network.Machine.Status.Clock07AdvStep),
i_rOnPosition		:= MC_InputOutput.Network.Machine.Parameters.Cam07OnValue,
i_rOffPosition		:= MC_InputOutput.Network.Machine.Parameters.Cam07OffValue,
i_rAdvanceTime		:= MC_InputOutput.Network.Machine.Parameters.Cam07AdvTime,
i_usiNumberOfPulse	:= MC_InputOutput.Network.Machine.Parameters.Cam07Pulse,
);

fbCam08(
i_xEnable			:= TRUE,
i_pxPointerOutput	:= ADR(MC_InputOutput.Network.Machine.Status.Clock08),
i_pxPointerStepAdv	:= ADR(MC_InputOutput.Network.Machine.Status.Clock08AdvStep),
i_rOnPosition		:= MC_InputOutput.Network.Machine.Parameters.Cam08OnValue,
i_rOffPosition		:= MC_InputOutput.Network.Machine.Parameters.Cam08OffValue,
i_rAdvanceTime		:= MC_InputOutput.Network.Machine.Parameters.Cam08AdvTime,
i_usiNumberOfPulse	:= MC_InputOutput.Network.Machine.Parameters.Cam08Pulse,
);

fbCam09(
i_xEnable			:= TRUE,
i_pxPointerOutput	:= ADR(MC_InputOutput.Network.Machine.Status.Clock09),
i_pxPointerStepAdv	:= ADR(MC_InputOutput.Network.Machine.Status.Clock09AdvStep),
i_rOnPosition		:= MC_InputOutput.Network.Machine.Parameters.Cam09OnValue,
i_rOffPosition		:= MC_InputOutput.Network.Machine.Parameters.Cam09OffValue,
i_rAdvanceTime		:= MC_InputOutput.Network.Machine.Parameters.Cam09AdvTime,
i_usiNumberOfPulse	:= MC_InputOutput.Network.Machine.Parameters.Cam09Pulse,
);

fbCam10(
i_xEnable			:= TRUE,
i_pxPointerOutput	:= ADR(MC_InputOutput.Network.Machine.Status.Clock10),
i_pxPointerStepAdv	:= ADR(MC_InputOutput.Network.Machine.Status.Clock10AdvStep),
i_rOnPosition		:= MC_InputOutput.Network.Machine.Parameters.Cam10OnValue,
i_rOffPosition		:= MC_InputOutput.Network.Machine.Parameters.Cam10OffValue,
i_rAdvanceTime		:= MC_InputOutput.Network.Machine.Parameters.Cam10AdvTime,
i_usiNumberOfPulse	:= MC_InputOutput.Network.Machine.Parameters.Cam10Pulse,
);

fbCam11(
i_xEnable			:= CFG_Par.Doser.Present,  //v999 test
i_pxPointerOutput	:= ADR(MC_InputOutput.Network.Machine.Status.Clock11),
i_pxPointerStepAdv	:= ADR(MC_InputOutput.Network.Machine.Status.Clock11AdvStep),
i_rOnPosition		:= MC_InputOutput.Network.Machine.Parameters.Cam11OnValue,
i_rOffPosition		:= MC_InputOutput.Network.Machine.Parameters.Cam11OffValue,
i_rAdvanceTime		:= MC_InputOutput.Network.Machine.Parameters.Cam11AdvTime,
i_usiNumberOfPulse	:= MC_InputOutput.Network.Machine.Parameters.Cam11Pulse,
);
END_STEP
TRANSITION ReturnToInitCondition FROM (FbMaster,CamMasterManagement,CamFb) TO Init:=
//V4.A.A.1.6.12d

(NOT VAR_Machine.stInletModule.iq_stStatus.q_xInitDone AND VAR_Machine.stInletModule.iq_stStatus.q_xModuleReal) OR
(NOT VAR_Machine.stFillerModule.iq_stStatus.q_xInitDone AND VAR_Machine.stFillerModule.iq_stStatus.q_xModuleReal) OR
(NOT VAR_Machine.stOutletModule.iq_stStatus.q_xInitDone AND VAR_Machine.stOutletModule.iq_stStatus.q_xModuleReal)
END_TRANSITION
(* @SFCISJUMP := 'Init' *)
END_PROGRAM
```

### Program Logical/30_MC/Task/Cyclic02/MC_MACHINE (IEC) - MC_MACHINE - C#1 0.8ms or C#2 10.4ms
